FUNCTION_BLOCK FB_AuditLog
VAR
	Event						 : FB_TcMessage;
	JsonParser					 : FB_JsonDomParser;
	TimeFormatter				 : FB_FormatString;
	MessagesSentThisScan		 : UDINT;
	Previous_k	 				 : T_MaxString;
	Previous_v					 : T_MaxString;
	InitComplete				 : BOOL := FALSE;
END_VAR

//FB_Init is always available implicitly and it is used primarily for initialization.
//The return value is not evaluated. For a specific influence, you can also declare the
//methods explicitly and provide additional code there with the standard initialization
//code. You can evaluate the return value.
METHOD FB_Init: BOOL
VAR_INPUT
    bInitRetains: BOOL; // TRUE: the retain variables are initialized (reset warm / reset cold)
    bInCopyCode: BOOL;  // TRUE: the instance will be copied to the copy code afterward (online change)   
END_VAR

VAR
	hr : HRESULT;
END_VAR
//	IF SUCCEEDED(Event.CreateEx(TC_EVENTS.Tracing.TraceEvent, 0)) THEN
{analysis -15}
IF ( NOT Event.EqualsToEventEntryEx(TC_EVENTS.Tracing.TraceEvent) ) THEN
	IF ( SUCCEEDED(Event.CreateEx(TC_EVENTS.AuditLog.Logger, 0)) ) THEN
		initComplete := TRUE;
	END_IF
ELSE
	initComplete := TRUE;
END_IF
END_METHOD

METHOD PRIVATE M_AddContext

VAR_INPUT
	json 			: SJsonValue;
	k 				: REFERENCE TO T_MaxString;
	v 				: REFERENCE TO T_MaxString;
END_VAR

VAR
	// Time 
	currentDCTime 			: DCTIMESTRUCT;
	task 					: T_MaxString;
	cycleCount 				: UDINT;
	msg						: STRING(255);
END_VAR
//Collect Properties
currentDCTime := DCTIME64_TO_DCTIMESTRUCT(F_GetActualDcTime64());
TimeFormatter(
    sFormat := '%2.2d:%2.2d:%2.2d.%3.3d%3.3d',
    arg1    := F_WORD(currentDCTime.wHour),
    arg2    := F_WORD(currentDCTime.wMinute),
    arg3    := F_WORD(currentDCTime.wSecond),
    arg4    := F_WORD(currentDCTime.wMilliseconds),
    arg5    := F_WORD(currentDCTime.wMicroseconds),	
    bError  => ,    // If there's a formatting error, this is TRUE
    nErrId  =>      // Error ID if bError=TRUE
);		
msg := CONCAT(k,v);
Event.ipArguments.Clear().AddString(msg);

// Pass properties to Json extnsion for logging.
jsonParser.AddStringMember(json, 'Timestamp', timeFormatter.sOut);
jsonParser.AddStringMember(json, 'k', k);
jsonParser.AddStringMember(json, 'v', v);
END_METHOD

METHOD M_AddEntry : BOOL
VAR_INPUT
	k 					: T_MaxString;
	v 					: T_MaxString;
END_VAR

VAR
	document	  		: SJsonValue;
	jsonAttribute 		: T_MaxString;
END_VAR
IF ( NOT InitComplete ) THEN
	RETURN;
END_IF

{analysis -62}
IF ( NOT pTracingAllowed ) THEN
	{analysis -90}
	RETURN;
END_IF

IF ( NOT Parameters_Tracing.ALLOW_DUPLICATE_SEQUENTIAL_MESSAGES ) THEN
	IF ( (k = Previous_k) AND (v = Previous_v) ) THEN
		//This message is identical to the last message sent--ignore
		RETURN;
	END_IF
END_IF

// Create JSON, add Context and add to Event
document := JsonParser.NewDocument();
M_AddContext(JSON := Document, k := k, v := v);
jsonAttribute := JsonParser.GetJson(document);
event.SetJsonAttribute(jsonAttribute);

// Send Event
Event.Send(0);

// Tidy up
MessagesSentThisScan := MessagesSentThisScan + 1;
MEMSET(ADR(Previous_k), 0, SIZEOF(T_MaxString));
MEMSET(ADR(Previous_v), 0, SIZEOF(T_MaxString));
Previous_k	 := k;
Previous_v := v;
END_METHOD

PROPERTY pTracingAllowed : BOOL
GET
VAR_INST
	LastScanCount  : UDINT;
	MissedMessages : UDINT;
	Throttled	   : BOOL;
END_VAR

VAR
	ThrottledNotificationString : T_MaxString;
END_VAR
{analysis -62}
IF NOT Parameters_Tracing.TRACING_ENABLED THEN
	pTracingAllowed := FALSE;
	RETURN;
END_IF

IF TwinCAT_SystemInfoVarList._TaskInfo[GETCURTASKINDEXEX()].CycleCount = LastScanCount THEN
	//Trying to send multiple messages in same scan
	IF Throttled THEN
		MissedMessages := MissedMessages + 1;
		RETURN;
	ELSIF MessagesSentThisScan >= Parameters_Tracing.MAX_LOG_ENTRIES_PER_SCAN AND NOT Throttled THEN
		//Need to throttle messsage queue
		Event.ipArguments.Clear().AddString('Too many messages sent in single scan; tracing throttled.');
		Event.Send(0);
		MissedMessages := MissedMessages + 1;
		Throttled	   := TRUE;
		pTracingAllowed := FALSE;
		RETURN;
	ELSE
		pTracingAllowed := TRUE;
	END_IF
ELSE
	IF Throttled THEN
		ThrottledNotificationString := CONCAT('Missed ', CONCAT(TO_STRING(MissedMessages), ' throttled messages previously.'));
		Event.ipArguments.Clear().AddString(ThrottledNotificationString);
		Event.Send(0);
		MissedMessages := 0;
	END_IF

	LastScanCount		 := TwinCAT_SystemInfoVarList._TaskInfo[GETCURTASKINDEXEX()].CycleCount;
	MessagesSentThisScan := 0;
	Throttled			 := FALSE;
	pTracingAllowed		 := TRUE;
END_IF
END_GET
END_PROPERTY

END_FUNCTION_BLOCK

(* stored: Version 1.1.0.1
   POU FB_AuditLog: Id {9f088aee-3833-491d-b09c-e2687a7d2630}, SpecialFunc None
   Method FB_Init: Id {7a89f529-4923-4ae2-917a-ed5d3a9b919e}
   Method M_AddContext: Id {664b27c4-60b4-47a0-9fcc-9f0b74dbbeaa}
   Method M_AddEntry: Id {6ccfe731-776e-42d3-b521-560e7cca4c70}
   Property pTracingAllowed: Id {b8050e1e-9d62-4288-a7ee-f696f5b0585d}
   Get Get: Id {9d392c52-98fa-4ba7-84a1-7da360ec224c} *)
